FUNCTION_BLOCK MachineSequenceStop EXTENDS MachineSequence IMPLEMENTS ZCore.ISequence
VAR
  _step : ZCore.Step(MachineStep.StopBegin, MachineStep.StopEnd);
  _timerSim : ZAux.Timer;
END_VAR

IF OnStart(_step) THEN
  ; // init custom sequence variables here ...
END_IF

REPEAT
  LogStep();

  CASE _step.Index OF
    (* -------------------------------------------------------------------------------------------------------------------------------- *)
    MachineStep.StopBegin:
    (* -------------------------------------------------------------------------------------------------------------------------------- *)
      IF _step.OnEntry()
      THEN
        _unit.PrimaryGear.StopAsync(THIS^, _parent);
        _unit.SimpleGear.StopAsync(THIS^, _parent);     
        _unit.StruckigGear.StopAsync(THIS^, _parent);           
      END_IF
      
      Await3(_unit.PrimaryGear, _unit.SimpleGear, _unit.StruckigGear, nextStep:=MachineStep.StopEnd);

    (* -------------------------------------------------------------------------------------------------------------------------------- *)
    MachineStep.StopEnd:
    (* -------------------------------------------------------------------------------------------------------------------------------- *)    
      SetBusy(FALSE);
  
  ELSE
    Abort('sequence contains unhandled step');
  END_CASE
UNTIL _step.IsNotRepeatable() OR_ELSE NOT Busy END_REPEAT

END_FUNCTION_BLOCK

(* stored: Version 1.1.0.1
   POU MachineSequenceStop: Id {a530cd4b-83ad-440c-84b4-af6f430a5012}, SpecialFunc None *)
